VISUALIZATION log_file  // 2x2
END_VISUALIZATION

(* stored: Version 1.1.0.1, ProductVersion 3.1.4024.12
   Visu log_file: Id {ae64ca54-3639-4de1-93f1-6e048eb65695} *)
